PROGRAM MAIN
VAR
	pneuma: FB_Pneumatic(enDB := FALSE);
	state: INT;
END_VAR


pneuma();

CASE state OF
	5:
		IF pneuma.doWait() THEN
			state := 0;
		END_IF
	10:
		IF pneuma.doWork() THEN
			state := 0;
		END_IF
END_CASE

END_PROGRAM

(* stored: Version 1.1.0.1, ProductVersion 3.1.4024.10
   POU MAIN: Id {d7f103ab-3e25-427e-8317-c3ab179e225d}, SpecialFunc None *)
